ABB RobotStudio station: p2_celula_pick&place_R2022_20231025-134356.rsstn

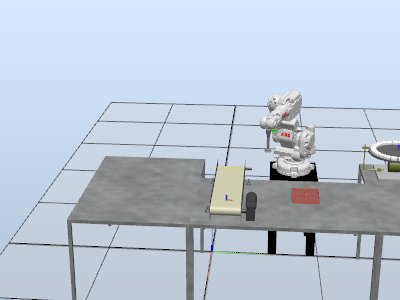
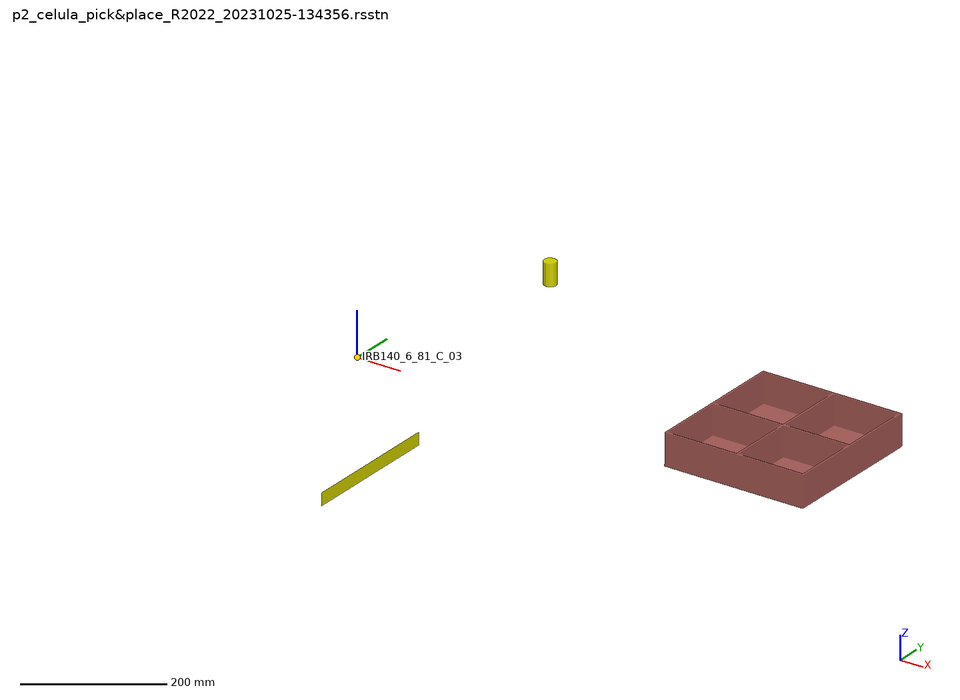
[picture v1: parts stored in the station drawn from their meshes, with robot base, taught points and paths (robot models come from the ABB library and are not in the file)]
Station p2_celula_cinta_mesagir_RS2019_2122_v2 (saved by RobotStudio 22.2.10013.1)
Controller Controlador1, task T_ROB1: task frame (RAPID world) sits at (-250, 750, 760) mm in the station
Controller Controlador1
  mechanical unit ROB_1: IRB140_6_81_C_03, 6 joints, base frame (0, 0, 0) mm
Layout (positions relative to the parent item):
  - Mesa de trabajo [part, from p2_RobotStudio\Mesa de trabajo.rslib] at (1000, -110, 0) mm, rotated rx 0 ry 0 rz 90 deg
  - Soporte [part, from p2_RobotStudio\SoporteDISA.rslib] at (-500, 970, 0) mm
  - Mesa giratoria [mechanism, from p2_RobotStudio\CAD Mesa giratoria.rslib] at (-400, 1510, 760) mm; joint values [1.5268] (rad or m)
  - Mesa de trabajo_2 [part, from p2_RobotStudio\Mesa de trabajo_2.rslib] at (1000, 2390, 0) mm, rotated rx 0 ry 0 rz 180 deg
  - cinta_transportadora [smart component, from p2_RobotStudio\cinta_transportadoraDISA_RI_vf.rslib]
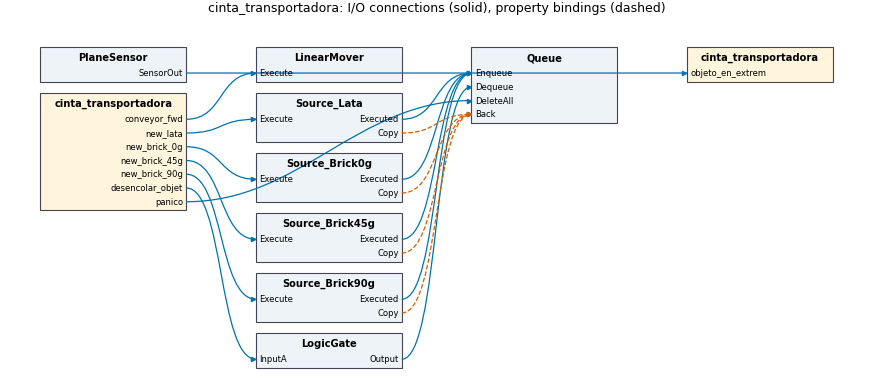
      connections:
        Source_Lata.Executed -> Queue.Enqueue
        PlaneSensor.SensorOut -> cinta_transportadora.objeto_en_extremo
        LogicGate.Output -> Queue.Dequeue
        cinta_transportadora.conveyor_fwd -> LinearMover.Execute
        cinta_transportadora.new_lata -> Source_Lata.Execute
        cinta_transportadora.new_brick_0g -> Source_Brick0g.Execute
        Source_Brick0g.Executed -> Queue.Enqueue
        cinta_transportadora.new_brick_45g -> Source_Brick45g.Execute
        Source_Brick45g.Executed -> Queue.Enqueue
        cinta_transportadora.new_brick_90g -> Source_Brick90g.Execute
        Source_Brick90g.Executed -> Queue.Enqueue
        cinta_transportadora.desencolar_objeto -> LogicGate.InputA
        cinta_transportadora.panico -> Queue.DeleteAll
        Source_Lata.Copy => Queue.Back
        Source_Brick0g.Copy => Queue.Back
        Source_Brick45g.Copy => Queue.Back
        Source_Brick90g.Copy => Queue.Back
    - Cinta transportadora [mechanism, from p2_RobotStudio\CAD Cinta transportadora_2.rslib] at (940, 100, 865) mm, rotated rx 0 ry 0 rz 90 deg; joint values [0.66] (rad or m)
    - PlaneSensor [smart component, from Components\PlaneSensor.rslib]
        properties: Origin=[0.17366 0.29 0.93]; Axis1=[0 -0.23 0]; Axis2=[0 0 0.02]; SensedPart=(none)
      - _sensorPart_ [part], size 0 x 230 x 20 mm
    - Source_Lata [smart component, from Components\Source.rslib]
        properties: Source=lata_v3; Copy=(none); Parent=(none); Position=[0.9 0.175 0.9]; Orientation=[0 0 0]; Transient=false; PhysicsBehavior=0
    - Queue [smart component, from Components\Queue.rslib]
        properties: Back=(none); Front=(none); Queue={57c4b1d3-0309-4464-8a6a-2fe5b6e73500};{5aa46dc6-d55b-4b09-bf64-be18c163c72f};{cdef8f33-6c1f-4f39-8898-60fe13adcf48};{42960cd8-682e-402a-8aab-2d8c8713f621};{119e90eb-0f41-47b6-a7f2-1fe2ae313f7f};{2b765b4e-81db-4cc5-9dbe-bde5ca058292};{dc2e37a3-00af-4aaa-b15c-731766a0f7c7};{3cac4617-f299-46fb-a085-5a6cb51f5200};{7a66cae6-64c5-4ef7-b2d4-279237335e64};{279f7df3-202b-4aa6-9977-3163501259bb};{f6008109-f320-423e-889e-dbc8c240ad71};{871d414f-ddac-4185-94d4-ee19182f4be7};{c4a57190-5175-4591-82fe-ecf9dac6460a};{3089afbe-ece1-4081-937c-81badaa6ba10};{e1825430-4c5a-4d9d-a921-2c138d7f3b2b};{7d8b643c-892a-4918-bfbd-a325ccae9b08};{0376169a-0871-4210-ba59-8bf384168a72};{59dac383-7526-4166-bc53-2ff7f1eed418};{174a4c52-5189-4e0a-a952-24ba83843141};{c153693b-fd65-4158-aa81-6a521c4dcca4};{1ab04711-27c4-4a9d-975f-98727157ab1c};{ff8ce740-4c14-42cd-a83a-c605c081d066};{0a6740bd-82d1-4125-b06b-8b1425ae5d33};{4edf2f45-6f83-4abc-bce2-8a18ddf87a8a};{0b049374-3d69-441a-9cbf-2320dfa0b1e3}; NumberOfObjects=1
    - LogicGate [smart component, from Components\LogicGate.rslib]
        properties: Operator=NOT; Delay=0
    - LinearMover [smart component, from Components\LinearMover.rslib]
        properties: Object=Queue; Direction=[1 0 0]; Speed=-0.5; Reference=Global; ReferenceObject=(none)
    - Source_Brick0g [smart component, from Components\Source.rslib]
        properties: Source=Brick0g; Copy=(none); Parent=(none); Position=[0.7 0.13 0.9]; Orientation=[0 0 0]; Transient=false; PhysicsBehavior=0
    - Source_Brick45g [smart component, from Components\Source.rslib]
        properties: Source=Brick0g; Copy=(none); Parent=(none); Position=[0.77 0.08 0.9]; Orientation=[0 0 0.785398163397448]; Transient=false; PhysicsBehavior=0
    - Source_Brick90g [smart component, from Components\Source.rslib]
        properties: Source=Brick0g; Copy=(none); Parent=(none); Position=[0.93 0.065 0.9]; Orientation=[0 0 1.5707963267949]; Transient=false; PhysicsBehavior=0
  - Brick0g [part, from p2_RobotStudio\Brick0g.rslib] at (332.58, -31.02, 436.47) mm
  - lata_v3 [part, from p2_RobotStudio\lata_v3.rslib] at (0.05, -0.04, 0.75) mm, rotated rx 0 ry 0 rz 0.02 deg
  - Pieza_11 [part], size 231 x 233 x 51.1 mm
  - Mesa de trabajo_3 [part, from p2_RobotStudio\Mesa de trabajo_3.rslib] at (1000, -110, 0) mm, rotated rx 0 ry 0 rz 180 deg
  - ventosa_giu [smart component, from p2_RobotStudio\ventosa_DISA_RI.rslib] at (245, 500, 1320) mm, rotated rx 180 ry 0 rz -180 deg
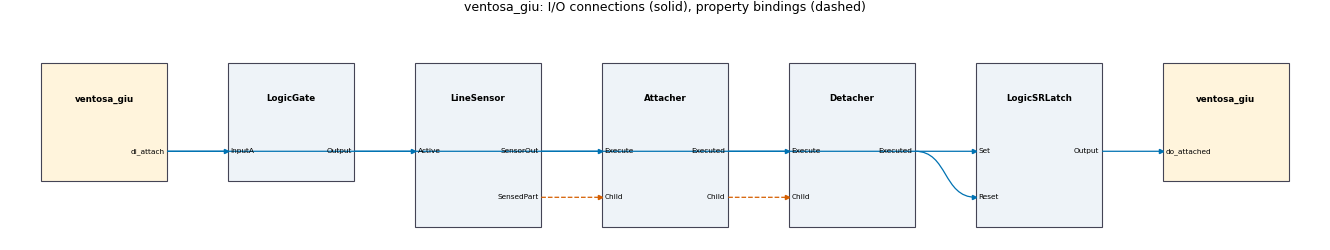
      connections:
        ventosa_giu.di_attach -> LogicGate.InputA
        LineSensor.SensorOut -> Attacher.Execute
        LogicGate.Output -> LineSensor.Active
        ventosa_giu.di_attach -> Detacher.Execute
        Attacher.Executed -> LogicSRLatch.Set
        Detacher.Executed -> LogicSRLatch.Reset
        LogicSRLatch.Output -> ventosa_giu.do_attached
        LineSensor.SensedPart => Attacher.Child
        Attacher.Child => Detacher.Child
    - ventosa_disa_giu [part, from p2_RobotStudio\ventosa_DISA_RI.rslib]
    - LogicGate [smart component, from Components\LogicGate.rslib]
        properties: Operator=NOT; Delay=0
    - LineSensor [smart component, from Components\LineSensor.rslib]
        properties: Start=[0 0 0.175]; End=[0 0 0.21]; Radius=0.01; SensedPart=(none); SensedPoint=[0.262718109130859 0.48144189453125 1.10501330566406]
      - _sensorPart_ [part], size 20 x 20 x 35 mm
    - Attacher [smart component, from Components\Attacher.rslib]
        properties: Parent=ventosa_giu; Flange=0; Child=(none); Mount=false; Offset=[0 0 0]; Orientation=[0 0 0]
    - Detacher [smart component, from Components\Detacher.rslib]
        properties: Child=(none); KeepPosition=true
    - LogicSRLatch [smart component, from Components\LogicSRLatch.rslib]
  - IRB140_6_81_C_03 [mechanism, from Robots\IRB140_6_81_C_G_03.rslib] at (-250, 750, 760) mm; joint values [-0.4677, 0.3133, -0.1294, 0, 1.3869, -0.4677] (rad or m)
Attachment: ventosa_giu is attached to IRB140_6_81_C_03 / Link6
EventTableEntry 9242: Group=, Trigger=Abrir 9243, Actions=[EventTableActionNothing 12035, EventTableActionDetach 12036, EventTableActionDetach 12037, EventTableActionDetach 12038, EventTableActionDetach 12039, EventTableActionDetach 12040, EventTableActionDetach 12041], Comment=, ActivationMode=2, Cyclic=true
EventTableTriggerIO 9243: IOValue=[1], IRC5Controller=? -1, Operator=0, SignalSource=? -1
EventTableEntry 9251: Group=, Trigger=Cerrar 9252, Actions=[EventTableActionDetach 12042, EventTableActionDetach 12043, EventTableActionDetach 12044, EventTableActionDetach 12045, EventTableActionDetach 12046, EventTableActionDetach 12047, EventTableActionNothing 12048], Comment=, ActivationMode=2, Cyclic=true
EventTableTriggerIO 9252: IOValue=[1], IRC5Controller=? -1, Operator=0, SignalSource=? -1
EventTableEntry 9264: Group=, Trigger=NOP 9265, Actions=[Abrir 9267], Comment=, ActivationMode=2, Cyclic=false
EventTableTriggerLogic 9265: Operand1=DoGARRAOPEN 9266, Operand2=? -1, Operator=4, Delay=1000
EventTableTriggerIO 9266: IOValue=[-1], IRC5Controller=? -1, Operator=0, SignalSource=? -1
EventTableActionIO 9267: IOValue=[-1], IRC5Controller=? -1, SignalTarget=? -1
EventTableEntry 9268: Group=, Trigger=NOT 9269, Actions=[Cerrar 9271], Comment=, ActivationMode=2, Cyclic=false
EventTableTriggerLogic 9269: layoutX=105, layoutY=91, Operand1=DoGARRAOPEN 9270, Operand2=? -1, Operator=2, Delay=1000
EventTableTriggerIO 9270: IOValue=[-1], IRC5Controller=? -1, Operator=0, SignalSource=? -1
EventTableActionIO 9271: IOValue=[-1], IRC5Controller=? -1, SignalTarget=? -1
EventTableEntry 9272: Group=, Trigger=DoGARRAOPEN 9273, Actions=[EventTableActionMechanicalPose 9274], Comment=, ActivationMode=2, Cyclic=false
EventTableTriggerIO 9273: IOValue=[1], IRC5Controller=? -1, Operator=0, SignalSource=? -1
EventTableActionMechanicalPose 9274: VirtualSignal=, Mechanism=? -1, ToPoseName=Abierta, VirtualSignalValue=[1]
EventTableEntry 9275: Group=, Trigger=DoGARRAOPEN 9276, Actions=[EventTableActionMechanicalPose 9277], Comment=, ActivationMode=2, Cyclic=false
EventTableTriggerIO 9276: IOValue=[0], IRC5Controller=? -1, Operator=0, SignalSource=? -1
EventTableActionMechanicalPose 9277: VirtualSignal=, Mechanism=? -1, ToPoseName=Cerrada, VirtualSignalValue=[1]
EventTableEntry 9288: Group=, Trigger=DO10_4 9289, Actions=[EventTableActionMechanicalPose 10691, EventTableActionMechanicalPose 10690, EventTableActionMechanicalPose 10689, EventTableActionMechanicalPose 11250, EventTableActionMechanicalPose 11251, EventTableActionMechanicalPose 11252], Comment=, ActivationMode=2, Cyclic=true
EventTableTriggerIO 9289: IOValue=[1], IRC5Controller=? -1, Operator=0, SignalSource=? -1
EventTableEntry 9711: Group=, Trigger=Abrir 9712, Actions=[EventTableActionNothing 12049, EventTableActionAttach 12050, EventTableActionAttach 12051, EventTableActionAttach 12052, EventTableActionNothing 12053, EventTableActionNothing 12054, EventTableActionNothing 12055], Comment=, ActivationMode=2, Cyclic=true
EventTableTriggerIO 9712: IOValue=[1], IRC5Controller=? -1, Operator=0, SignalSource=? -1
EventTableEntry 9938: Group=, Trigger=Cerrar 9939, Actions=[EventTableActionAttach 12056, EventTableActionAttach 12057, EventTableActionAttach 12058, EventTableActionAttach 12059, EventTableActionAttach 12060, EventTableActionAttach 12061, EventTableActionNothing 12062], Comment=, ActivationMode=2, Cyclic=true
EventTableTriggerIO 9939: IOValue=[1], IRC5Controller=? -1, Operator=0, SignalSource=? -1
EventTableActionMechanicalPose 10689: VirtualSignal=, Mechanism=Mesa giratoria 10339, ToPoseName=360º, VirtualSignalValue=[1]
EventTableActionMechanicalPose 10690: VirtualSignal=, Mechanism=Mesa giratoria 10339, ToPoseName=180º, VirtualSignalValue=[1]
EventTableActionMechanicalPose 10691: VirtualSignal=, Mechanism=Mesa giratoria 10339, ToPoseName=90º, VirtualSignalValue=[1]
EventTableEntry 11031: Group=, Trigger=DO10_5 11032, Actions=[EventTableActionAttach 11212, EventTableActionAttach 11213, EventTableActionAttach 11214], Comment=, ActivationMode=2, Cyclic=true
EventTableTriggerIO 11032: IOValue=[1], IRC5Controller=? -1, Operator=0, SignalSource=? -1
EventTableEntry 11051: Group=, Trigger=Abrir 11052, Actions=[EventTableActionNothing 12063, EventTableActionMechanicalPose 12064, EventTableActionMechanicalPose 12065, EventTableActionNothing 12066, EventTableActionNothing 12067, EventTableActionNothing 12068, EventTableActionNothing 12069], Comment=, ActivationMode=2, Cyclic=true
EventTableTriggerIO 11052: IOValue=[1], IRC5Controller=? -1, Operator=0, SignalSource=? -1
EventTableEntry 11203: Group=, Trigger=DO10_5 11204, Actions=[EventTableActionMechanicalPose 11205, EventTableActionMechanicalPose 11206, EventTableActionMechanicalPose 11207], Comment=, ActivationMode=2, Cyclic=true
EventTableTriggerIO 11204: IOValue=[1], IRC5Controller=? -1, Operator=0, SignalSource=? -1
EventTableActionMechanicalPose 11205: VirtualSignal=, Mechanism=Cinta transportadora 10989, ToPoseName=HomePosition, VirtualSignalValue=[1]
EventTableActionMechanicalPose 11206: VirtualSignal=, Mechanism=Cinta transportadora 10989, ToPoseName=HomePosition, VirtualSignalValue=[1]
EventTableActionMechanicalPose 11207: VirtualSignal=, Mechanism=Cinta transportadora 10989, ToPoseName=HomePosition, VirtualSignalValue=[1]
EventTableActionAttach 11212: AttachmentParent=Cinta transportadora 10989, AttachmentChild=? -1, MountObject=false, Offset=[X=1, Y=0, Z=0, W=0, X=0, Y=1, Z=0, W=0, X=0, Y=0, Z=1, W=0, X=0, Y=0, Z=0, W=1], FlangeIndext=0, FindNearest=false
EventTableActionAttach 11213: AttachmentParent=Cinta transportadora 10989, AttachmentChild=? -1, MountObject=false, Offset=[X=1, Y=0, Z=0, W=0, X=0, Y=1, Z=0, W=0, X=0, Y=0, Z=1, W=0, X=0, Y=0, Z=0, W=1], FlangeIndext=0, FindNearest=false
EventTableActionAttach 11214: AttachmentParent=Cinta transportadora 10989, AttachmentChild=? -1, MountObject=false, Offset=[X=1, Y=0, Z=0, W=0, X=0, Y=1, Z=0, W=0, X=0, Y=0, Z=1, W=0, X=0, Y=0, Z=0, W=1], FlangeIndext=0, FindNearest=false
EventTableActionMechanicalPose 11250: VirtualSignal=, Mechanism=Mesa giratoria 10339, ToPoseName=450, VirtualSignalValue=[1]
EventTableActionMechanicalPose 11251: VirtualSignal=, Mechanism=Mesa giratoria 10339, ToPoseName=540º, VirtualSignalValue=[1]
EventTableActionMechanicalPose 11252: VirtualSignal=, Mechanism=Mesa giratoria 10339, ToPoseName=SyncPosition, VirtualSignalValue=[1]
EventTableEntry 11270: Group=, Trigger=DO10_6 11271, Actions=[EventTableActionAttach 11272, EventTableActionAttach 11273, EventTableActionAttach 11274], Comment=, ActivationMode=2, Cyclic=true
EventTableTriggerIO 11271: IOValue=[1], IRC5Controller=? -1, Operator=0, SignalSource=? -1
EventTableActionAttach 11272: AttachmentParent=Cinta transportadora 10989, AttachmentChild=? -1, MountObject=false, Offset=[X=1, Y=0, Z=0, W=0, X=0, Y=1, Z=0, W=0, X=0, Y=0, Z=1, W=0, X=0, Y=0, Z=0, W=1], FlangeIndext=0, FindNearest=false
EventTableActionAttach 11273: AttachmentParent=Cinta transportadora 10989, AttachmentChild=? -1, MountObject=false, Offset=[X=1, Y=0, Z=0, W=0, X=0, Y=1, Z=0, W=0, X=0, Y=0, Z=1, W=0, X=0, Y=0, Z=0, W=1], FlangeIndext=0, FindNearest=false
EventTableActionAttach 11274: AttachmentParent=Cinta transportadora 10989, AttachmentChild=? -1, MountObject=false, Offset=[X=1, Y=0, Z=0, W=0, X=0, Y=1, Z=0, W=0, X=0, Y=0, Z=1, W=0, X=0, Y=0, Z=0, W=1], FlangeIndext=0, FindNearest=false
EventTableEntry 11487: Group=, Trigger=Cerrar 11488, Actions=[EventTableActionNothing 12070, EventTableActionNothing 12071, EventTableActionNothing 12072, EventTableActionNothing 12073, EventTableActionMechanicalPose 12074, EventTableActionMechanicalPose 12075, EventTableActionNothing 12076], Comment=, ActivationMode=2, Cyclic=true
EventTableTriggerIO 11488: IOValue=[1], IRC5Controller=? -1, Operator=0, SignalSource=? -1
EventTableEntry 11751: Group=, Trigger=Cerrar 11752, Actions=[EventTableActionNothing 12077, EventTableActionNothing 12078, EventTableActionNothing 12079, EventTableActionNothing 12080, EventTableActionDetach 12081, EventTableActionDetach 12082, EventTableActionDetach 12083], Comment=, ActivationMode=2, Cyclic=true
EventTableTriggerIO 11752: IOValue=[1], IRC5Controller=? -1, Operator=0, SignalSource=? -1
EventTableEntry 11847: Group=, Trigger=DO10_6 11848, Actions=[EventTableActionMechanicalPose 11849, EventTableActionMechanicalPose 11850, EventTableActionMechanicalPose 11851], Comment=, ActivationMode=2, Cyclic=true
EventTableTriggerIO 11848: IOValue=[1], IRC5Controller=? -1, Operator=0, SignalSource=? -1
EventTableActionMechanicalPose 11849: VirtualSignal=, Mechanism=Cinta transportadora 10989, ToPoseName=Final, VirtualSignalValue=[1]
EventTableActionMechanicalPose 11850: VirtualSignal=, Mechanism=Cinta transportadora 10989, ToPoseName=Final, VirtualSignalValue=[1]
EventTableActionMechanicalPose 11851: VirtualSignal=, Mechanism=Cinta transportadora 10989, ToPoseName=Final, VirtualSignalValue=[1]
EventTableActionNothing 12035: 
EventTableActionDetach 12036: AttachmentParent=? -1, AttachmentChild=? -1
EventTableActionDetach 12037: AttachmentParent=? -1, AttachmentChild=? -1
EventTableActionDetach 12038: AttachmentParent=? -1, AttachmentChild=? -1
EventTableActionDetach 12039: AttachmentParent=? -1, AttachmentChild=? -1
EventTableActionDetach 12040: AttachmentParent=? -1, AttachmentChild=? -1
EventTableActionDetach 12041: AttachmentParent=? -1, AttachmentChild=? -1
EventTableActionDetach 12042: AttachmentParent=Cinta transportadora 10989, AttachmentChild=? -1
EventTableActionDetach 12043: AttachmentParent=Cinta transportadora 10989, AttachmentChild=? -1
EventTableActionDetach 12044: AttachmentParent=Cinta transportadora 10989, AttachmentChild=? -1
EventTableActionDetach 12045: AttachmentParent=Mesa giratoria 10339, AttachmentChild=? -1
EventTableActionDetach 12046: AttachmentParent=Mesa giratoria 10339, AttachmentChild=? -1
EventTableActionDetach 12047: AttachmentParent=Mesa giratoria 10339, AttachmentChild=? -1
EventTableActionNothing 12048: 
EventTableActionNothing 12049: 
EventTableActionAttach 12050: AttachmentParent=Mesa giratoria 10339, AttachmentChild=? -1, MountObject=false, Offset=[X=1, Y=0, Z=0, W=0, X=0, Y=1, Z=0, W=0, X=0, Y=0, Z=1, W=0, X=0, Y=0, Z=0, W=1], FlangeIndext=0, FindNearest=false
EventTableActionAttach 12051: AttachmentParent=Mesa giratoria 10339, AttachmentChild=? -1, MountObject=false, Offset=[X=1, Y=0, Z=0, W=0, X=0, Y=1, Z=0, W=0, X=0, Y=0, Z=1, W=0, X=0, Y=0, Z=0, W=1], FlangeIndext=0, FindNearest=false
EventTableActionAttach 12052: AttachmentParent=Mesa giratoria 10339, AttachmentChild=? -1, MountObject=false, Offset=[X=1, Y=0, Z=0, W=0, X=0, Y=1, Z=0, W=0, X=0, Y=0, Z=1, W=0, X=0, Y=0, Z=0, W=1], FlangeIndext=0, FindNearest=false
EventTableActionNothing 12053: 
EventTableActionNothing 12054: 
EventTableActionNothing 12055: 
EventTableActionAttach 12056: AttachmentParent=? -1, AttachmentChild=? -1, MountObject=true, Offset=[X=1, Y=0, Z=0, W=0, X=0, Y=1, Z=0, W=0, X=0, Y=0, Z=1, W=0, X=0, Y=0, Z=0, W=1], FlangeIndext=0, FindNearest=false
EventTableActionAttach 12057: AttachmentParent=? -1, AttachmentChild=? -1, MountObject=true, Offset=[X=1, Y=0, Z=0, W=0, X=0, Y=1, Z=0, W=0, X=0, Y=0, Z=1, W=0, X=0, Y=0, Z=0, W=1], FlangeIndext=0, FindNearest=false
EventTableActionAttach 12058: AttachmentParent=? -1, AttachmentChild=? -1, MountObject=true, Offset=[X=1, Y=0, Z=0, W=0, X=0, Y=1, Z=0, W=0, X=0, Y=0, Z=1, W=0, X=0, Y=0, Z=0, W=1], FlangeIndext=0, FindNearest=false
EventTableActionAttach 12059: AttachmentParent=? -1, AttachmentChild=? -1, MountObject=true, Offset=[X=1, Y=0, Z=0, W=0, X=0, Y=1, Z=0, W=0, X=0, Y=0, Z=1, W=0, X=0, Y=0, Z=0, W=1], FlangeIndext=0, FindNearest=false
EventTableActionAttach 12060: AttachmentParent=? -1, AttachmentChild=? -1, MountObject=true, Offset=[X=1, Y=0, Z=0, W=0, X=0, Y=1, Z=0, W=0, X=0, Y=0, Z=1, W=0, X=0, Y=0, Z=0, W=1], FlangeIndext=0, FindNearest=false
EventTableActionAttach 12061: AttachmentParent=? -1, AttachmentChild=? -1, MountObject=true, Offset=[X=1, Y=0, Z=0, W=0, X=0, Y=1, Z=0, W=0, X=0, Y=0, Z=1, W=0, X=0, Y=0, Z=0, W=1], FlangeIndext=0, FindNearest=false
EventTableActionNothing 12062: 
EventTableActionNothing 12063: 
EventTableActionMechanicalPose 12064: VirtualSignal=, Mechanism=Cinta transportadora 10989, ToPoseName=Final_2, VirtualSignalValue=[1]
EventTableActionMechanicalPose 12065: VirtualSignal=, Mechanism=Cinta transportadora 10989, ToPoseName=Final_2, VirtualSignalValue=[1]
EventTableActionNothing 12066: 
EventTableActionNothing 12067: 
EventTableActionNothing 12068: 
EventTableActionNothing 12069: 
EventTableActionNothing 12070: 
EventTableActionNothing 12071: 
EventTableActionNothing 12072: 
EventTableActionNothing 12073: 
EventTableActionMechanicalPose 12074: VirtualSignal=, Mechanism=Cinta transportadora 10989, ToPoseName=Pose inicial_2, VirtualSignalValue=[1]
EventTableActionMechanicalPose 12075: VirtualSignal=, Mechanism=Cinta transportadora 10989, ToPoseName=Pose inicial_2, VirtualSignalValue=[1]
EventTableActionNothing 12076: 
EventTableActionNothing 12077: 
EventTableActionNothing 12078: 
EventTableActionNothing 12079: 
EventTableActionNothing 12080: 
EventTableActionDetach 12081: AttachmentParent=Cinta transportadora 10989, AttachmentChild=? -1
EventTableActionDetach 12082: AttachmentParent=Cinta transportadora 10989, AttachmentChild=? -1
EventTableActionDetach 12083: AttachmentParent=Cinta transportadora 10989, AttachmentChild=? -1
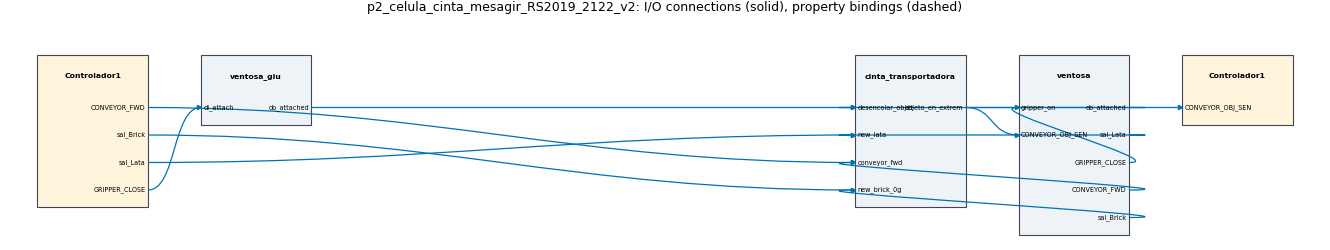
Station logic (signal -> signal, property => property):
  ventosa.do_attached -> cinta_transportadora.desencolar_objeto
  Controlador_P2_2021.sal_Lata -> cinta_transportadora.new_lata
  Controlador_P2_2021.GRIPPER_CLOSE -> ventosa.gripper_on
  cinta_transportadora.objeto_en_extremo -> Controlador_P2_2021.CONVEYOR_OBJ_SEN
  Controlador_P2_2021.CONVEYOR_FWD -> cinta_transportadora.conveyor_fwd
  Controlador_P2_2021.sal_Brick -> cinta_transportadora.new_brick_0g
  ventosa_giu.do_attached -> cinta_transportadora.desencolar_objeto
  Controlador1.CONVEYOR_FWD -> cinta_transportadora.conveyor_fwd
  Controlador1.sal_Brick -> cinta_transportadora.new_brick_0g
  Controlador1.sal_Lata -> cinta_transportadora.new_lata
  Controlador1.GRIPPER_CLOSE -> ventosa_giu.di_attach
  cinta_transportadora.objeto_en_extremo -> Controlador1.CONVEYOR_OBJ_SEN
